// TwinCAT 3 PLC project TcAdsExamplesPlcRt
// ProgramVersion: 3.1.4024.0
// libraries:
//   Tc2_Standard, * (Beckhoff Automation GmbH)
//   Tc2_System, * (Beckhoff Automation GmbH)
//   Tc2_Utilities, * (Beckhoff Automation GmbH)
//   Tc3_Module, * (Beckhoff Automation GmbH)
// project tree:
//   DUTs/ E_RecipeStepCommand.TcTLEO, ST_Empty.TcDUT, ST_RecipeStep.TcDUT, T_RecipeId.TcDUT, T_RecipeStep.TcDUT, T_STEmptyAlias.TcDUT
//   ITFs/ I_Empty.TcIO, I_EmptyWithExtends.TcIO, I_WithMethods.TcIO, I_WithMethodsPropsAndExtends.TcIO, I_WithProps.TcIO, I_WithRPC.TcIO
//   / PlcTask.TcTTO
//   POUs/FBs/ FB_EmptyWithRPC.TcPOU, FB_Empty.TcPOU, FB_EmptyWithExtends.TcPOU, FB_EmptyWithEmptyImpl.TcPOU, FB_EmptyWithImplRPC.TcPOU, FB_MathMachine.TcPOU, FB_Recipe.TcPOU, FB_WithFields.TcPOU
//   POUs/Fs/ F_ResetOnTrue.TcPOU
//   POUs/ MAIN.TcPOU, P_DataTypesExample.TcPOU
// real-time tasks:
//   TASK PlcTask: cycle T#10ms, priority 20, ADS port 350

CONFIGURATION TcAdsExamplesPlcRt
    RESOURCE PLC ON TwinCAT3
        TASK PlcTask(INTERVAL := T#10ms, PRIORITY := 20);
        PROGRAM MAIN WITH PlcTask : MAIN;
        PROGRAM P_DataTypesExample WITH PlcTask : P_DataTypesExample;
    END_RESOURCE
END_CONFIGURATION

// ---- DUTs/E_RecipeStepCommand.TcTLEO
{attribute 'qualified_only'}
{attribute 'strict'}
{attribute 'to_string'}
TYPE E_RecipeStepCommand :
(
	Idle := 0,
	Heat,
	Cool,
	Mix,
	Pump
)BYTE;
END_TYPE

// ---- DUTs/ST_Empty.TcDUT
TYPE ST_Empty :
STRUCT
END_STRUCT
END_TYPE

// ---- DUTs/ST_RecipeStep.TcDUT
TYPE ST_RecipeStep :
STRUCT
	eCommand 	: E_RecipeStepCommand;
	fTarget 	: LREAL;
	tDuration	: TIME;
END_STRUCT
END_TYPE

// ---- DUTs/T_RecipeId.TcDUT
TYPE T_RecipeId : STRING(20); END_TYPE

// ---- DUTs/T_RecipeStep.TcDUT
TYPE T_RecipeStep : ST_RecipeStep; END_TYPE

// ---- DUTs/T_STEmptyAlias.TcDUT
TYPE T_STEmptyAlias : ST_Empty; END_TYPE

// ---- ITFs/I_Empty.TcIO
// Basic empty interface, no inheritance, no methods no properties.
INTERFACE I_Empty

END_INTERFACE

// ---- ITFs/I_EmptyWithExtends.TcIO
// Empty interface that inherits an empty inteface.
INTERFACE I_EmptyWithExtends EXTENDS __SYSTEM.IQueryInterface

END_INTERFACE

// ---- ITFs/I_WithMethods.TcIO
// Interface with only methods
INTERFACE I_WithMethods

// A method with all types of input and outputs as well as a return type.
METHOD FullMethod : UDINT
VAR_INPUT
	InArg1  	: STRING(64);
	InArg2		: Tc2_System.ST_AmsAddr; 
END_VAR
VAR_IN_OUT
	InOutArg1	: POINTER TO __UXINT;
END_VAR
VAR_OUTPUT
	OutArg1		: Tc2_System.E_SeekOrigin;
	OutArg2		: Tc2_System.T_MaxString;
END_VAR
END_METHOD

// A method with only a return type an no args.
METHOD ReturnOnlyMethod : BOOL
VAR_INPUT
END_VAR
END_METHOD

// A method that has no arguments.
METHOD VoidMethod
VAR_INPUT
END_VAR
END_METHOD

END_INTERFACE

// ---- ITFs/I_WithMethodsPropsAndExtends.TcIO
// Interface with inheritence, methods and properties.
INTERFACE I_WithMethodsPropsAndExtends EXTENDS __SYSTEM.IQueryInterface

// A method with all types of input and outputs as well as a return type.
METHOD FullMethod : UDINT
VAR_INPUT
	InArg1  	: STRING(64);
	InArg2		: Tc2_System.ST_CpuCoreInfo; 
END_VAR
VAR_IN_OUT
	InOutArg1	: POINTER TO __UXINT;
END_VAR
VAR_OUTPUT
	OutArg1		: Tc2_System.E_SeekOrigin;
	OutArg2		: Tc2_System.T_MaxString;
END_VAR
END_METHOD

// First property.
PROPERTY Prop1 : BOOL
GET
END_GET
SET
END_SET
END_PROPERTY

// Second property.
PROPERTY Prop2 : Tc2_System.ST_CpuCoreInfo
GET
END_GET
SET
END_SET
END_PROPERTY

// A method with only a return type an no args.
METHOD ReturnOnlyMethod : BOOL
VAR_INPUT
END_VAR
END_METHOD

// A method that has no arguments.
METHOD VoidMethod
VAR_INPUT
END_VAR
END_METHOD

END_INTERFACE

// ---- ITFs/I_WithProps.TcIO
// Interface with properties only.
INTERFACE I_WithProps

// First property.
PROPERTY Prop1 : BOOL
GET
END_GET
SET
END_SET
END_PROPERTY

// Second property.
PROPERTY Prop2 : Tc2_System.ST_CpuCoreInfo
GET
END_GET
SET
END_SET
END_PROPERTY

END_INTERFACE

// ---- ITFs/I_WithRPC.TcIO
// Interface with properties only.
INTERFACE I_WithRPC

// A method with all types of input and outputs as well as a return type.
{attribute 'TcRpcEnable'}
METHOD FullMethod : UDINT
VAR_INPUT
	InArg1  	: STRING(64);
	InArg2		: Tc2_System.ST_CpuCoreInfo; 
END_VAR
VAR_IN_OUT
	InOutArg1	: POINTER TO __UXINT;
END_VAR
VAR_OUTPUT
	OutArg1		: Tc2_System.E_SeekOrigin;
	OutArg2		: Tc2_System.T_MaxString;
END_VAR
END_METHOD

// First property.
{attribute 'TcRpcEnable'}
PROPERTY Prop1 : BOOL
GET
END_GET
SET
END_SET
END_PROPERTY

// A method that has no arguments.
{attribute 'TcRpcEnable'}
METHOD VoidMethod
VAR_INPUT
END_VAR
END_METHOD

END_INTERFACE

// ---- POUs/MAIN.TcPOU
// This is an example TwinCAT Runtime project for tcads-rs demonstrations.
PROGRAM MAIN
VAR
	nCount 			: UDINT := 99;
	bIncrement 		: BOOL;
	bDecrement 		: BOOL;
	
	fbCurrentRecipe	: FB_Recipe;
	fbMath 			: FB_MathMachine;
END_VAR

IF F_ResetOnTrue(bIncrement) THEN 
	nCount := nCount + 1;
	ADSLOGSTR(
        msgCtrlMask := ADSLOG_MSGTYPE_WARN, 
        msgFmtStr   := 'Increment -> %s', 
        strArg      := TO_STRING(nCount)
    );
END_IF

IF F_ResetOnTrue(bDecrement) THEN 
	nCount := nCount - 1;
	ADSLOGSTR(
        msgCtrlMask := ADSLOG_MSGTYPE_ERROR, 
        msgFmtStr   := 'Decrement -> %s', 
        strArg      := TO_STRING(nCount)
    );
END_IF

END_PROGRAM

// ---- POUs/FBs/FB_Recipe.TcPOU
{attribute 'no_explicit_call' := 'direct call for this function block is not allowed'}
FUNCTION_BLOCK FB_Recipe IMPLEMENTS  __SYSTEM.IQueryInterface
VAR
	Id 		: T_RecipeId;
	arSteps : ARRAY[0..4] OF T_RecipeStep;
END_VAR

END_FUNCTION_BLOCK

// ---- POUs/FBs/FB_MathMachine.TcPOU
{attribute 'no_explicit_call' := 'direct call for this function block is not allowed'}
FUNCTION_BLOCK FB_MathMachine
VAR
	_nValue : DINT;
END_VAR

{attribute 'TcRpcEnable'}
METHOD DivideValues : DINT
VAR_INPUT
	nNumerator, 
	nDenominator : DINT;
END_VAR
VAR_OUTPUT
	nRemainder   : DINT;
END_VAR
IF nDenominator <> 0 THEN
	DivideValues := nNumerator / nDenominator;
	nRemainder   := nNumerator MOD nDenominator;
END_IF
END_METHOD

{attribute 'TcRpcEnable'}
METHOD GetValue : DINT
VAR_INPUT
END_VAR
GetValue := THIS^._nValue;
END_METHOD

{attribute 'TcRpcEnable'}
METHOD Reset
VAR_INPUT
END_VAR
 THIS^._nValue := 0;
END_METHOD

{attribute 'TcRpcEnable'}
METHOD SetValue
VAR_INPUT
	nValue : DINT;
END_VAR
THIS^._nValue := nValue;
END_METHOD

{attribute 'TcRpcEnable'}
METHOD SumValues : DINT
VAR_INPUT
	nValue1, nValue2 : DINT;
END_VAR
SumValues := nValue1 + nValue2;
END_METHOD

END_FUNCTION_BLOCK

// ---- POUs/Fs/F_ResetOnTrue.TcPOU
// Sets the boolean value to false if it is true and returns true if it was true before being set.
FUNCTION F_ResetOnTrue  : BOOL // Whether the value was true before resetting.
VAR_INPUT
	bValue : REFERENCE TO BOOL; // Boolean value to reset.
END_VAR

F_ResetOnTrue 	:= bValue;
bValue 			:= FALSE;

END_FUNCTION

// ---- POUs/P_DataTypesExample.TcPOU
// Contains varias TwinCAT Runtime datatypes for tcads-rs's DataTypeDevice
PROGRAM P_DataTypesExample
VAR
	// Interfaces
	
	ipEmpty 					: I_Empty;
	ipEmptyWithExtends 			: I_EmptyWithExtends;
	ipWithProps					: I_WithProps;
	ipWithMethods				: I_WithMethods;
	ipWithMethodPropsAndExtends : I_WithMethodsPropsAndExtends;
	ipWithRPC					: I_WithRPC;
	
	// Function Blocks
	
	fbEmpty 					: FB_Empty;
	fbEmptyWithExtends 			: FB_EmptyWithExtends;
	fbEmptyWithEmptyImpl		: FB_EmptyWithEmptyImpl;
	fbWithFields				: FB_WithFields;
	fbEmptyWithRPC 				: FB_EmptyWithRPC;
	fbEmptyWithImplRPC 			: FB_EmptyWithImplRPC;
	
	// Structs
	
	stEmpty						: ST_Empty;
	STEmptyAlias				: T_STEmptyAlias;	
END_VAR

END_PROGRAM

// ---- POUs/FBs/FB_Empty.TcPOU
// Empty function block with no fields, properties, methods, inheritance or interfaces.
FUNCTION_BLOCK FB_Empty
VAR
END_VAR

END_FUNCTION_BLOCK

// ---- POUs/FBs/FB_EmptyWithExtends.TcPOU
// Empty function block that extends an empty function block.
FUNCTION_BLOCK FB_EmptyWithExtends EXTENDS FB_Empty
VAR
END_VAR

END_FUNCTION_BLOCK

// ---- POUs/FBs/FB_EmptyWithEmptyImpl.TcPOU
// Empty function block that implements an empty interface only.
FUNCTION_BLOCK FB_EmptyWithEmptyImpl
IMPLEMENTS I_Empty
VAR
END_VAR

END_FUNCTION_BLOCK

// ---- POUs/FBs/FB_WithFields.TcPOU
FUNCTION_BLOCK FB_WithFields
VAR_INPUT
	InField1 	: INT;
	InField2 	: Tc2_System.ST_CpuCoreInfo;
	InField3 	: ARRAY[0..4] OF INT;
END_VAR
VAR_IN_OUT
	InOutField1 : TIME;
END_VAR
VAR_OUTPUT
	{attribute 'hello there' := '42'}
	OutField1 	: __UXINT;
	// This is a comment for OutField2!
	OutField2 	: Tc2_System.E_TcMemoryArea;
END_VAR
VAR
END_VAR

END_FUNCTION_BLOCK

// ---- POUs/FBs/FB_EmptyWithRPC.TcPOU
{attribute 'no_explicit_call' := 'direct call for this function block is not allowed'}
FUNCTION_BLOCK FINAL FB_EmptyWithRPC
VAR
END_VAR

// A method with all types of input and outputs as well as a return type.
{attribute 'TcRpcEnable'}
METHOD FullMethod : UDINT
VAR_INPUT
	InArg1  	: STRING(64);
	InArg2		: Tc2_System.ST_CpuCoreInfo; 
END_VAR
VAR_IN_OUT
	InOutArg1	: POINTER TO __UXINT;
END_VAR
VAR_OUTPUT
	OutArg1		: Tc2_System.E_SeekOrigin;
	OutArg2		: Tc2_System.T_MaxString;
END_VAR
END_METHOD

// First property.
{attribute 'TcRpcEnable'}
PROPERTY Prop1 : BOOL
GET
END_GET
SET
END_SET
END_PROPERTY

// A method that has no arguments.
{attribute 'TcRpcEnable'}
METHOD VoidMethod
VAR_INPUT
END_VAR
END_METHOD

END_FUNCTION_BLOCK

// ---- POUs/FBs/FB_EmptyWithImplRPC.TcPOU
{attribute 'no_explicit_call' := 'direct call for this function block is not allowed'}
FUNCTION_BLOCK FINAL FB_EmptyWithImplRPC
IMPLEMENTS I_WithRPC
VAR
END_VAR

// A method with all types of input and outputs as well as a return type.
{attribute 'TcRpcEnable'}
METHOD FullMethod : UDINT
VAR_INPUT
	InArg1  	: STRING(64);
	InArg2		: Tc2_System.ST_CpuCoreInfo; 
END_VAR
VAR_IN_OUT
	InOutArg1	: POINTER TO __UXINT;
END_VAR
VAR_OUTPUT
	OutArg1		: Tc2_System.E_SeekOrigin;
	OutArg2		: Tc2_System.T_MaxString;
END_VAR
END_METHOD

// First property.
{attribute 'TcRpcEnable'}
PROPERTY Prop1 : BOOL
GET
END_GET
SET
END_SET
END_PROPERTY

// A method that has no arguments.
{attribute 'TcRpcEnable'}
METHOD VoidMethod
VAR_INPUT
END_VAR
END_METHOD

END_FUNCTION_BLOCK
